FUNCTION_BLOCK AUI_UDINT_AX_SEL_AUI (* binary selection *)
  (* Standard: 61131-3; Classification: standard selection function; Description: Copyright (c) 2012 TU Wien ACIN, HR Agrartechnik GmbH This program and the accompanying materials are made available under the terms of the Eclipse Public License 2.0 which is available at https://www.eclipse.org/legal/epl-2.0/ SPDX-License-Identifier: EPL-2.0 *)
  (* Version 3.0, 2025-04-14, Patrick Aigner, changed package *)
  (* Version 1.0, 2012-03-25, Monika Wenger, TU Wien ACIN, initial API and implementation and/or initial documentation *)
  PACKAGE adapter::iec61131::selection;
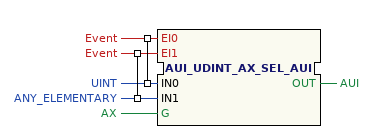
  EVENT_INPUT
    EI0 WITH IN0; (* Set IN0 *)
    EI1 WITH IN1; (* Set IN1 *)
  END_EVENT
  VAR_INPUT
    IN0 : UINT; (* Selectable input variable *)
    IN1 : ANY_ELEMENTARY; (* Selectable input variable *)
  END_VAR
  SOCKETS
    G : adapter::types::unidirectional::AX; (* Selelctor *)
  END_SOCKETS
  PLUGS
    OUT : adapter::types::unidirectional::AUI; (* Selected input *)
  END_PLUGS
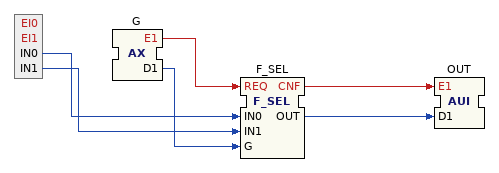
  FBS
    F_SEL : iec61131::selection::F_SEL;
  END_FBS
  EVENT_CONNECTIONS
    G.E1 TO F_SEL.REQ;
    F_SEL.CNF TO OUT.E1;
  END_CONNECTIONS
  DATA_CONNECTIONS
    IN0 TO F_SEL.IN0;
    IN1 TO F_SEL.IN1;
    G.D1 TO F_SEL.G;
    F_SEL.OUT TO OUT.D1;
  END_CONNECTIONS
END_FUNCTION_BLOCK
